Xinje XCPPro project, PLC1: XC3-24 (software 3.3L)

PROGRAM Ladder

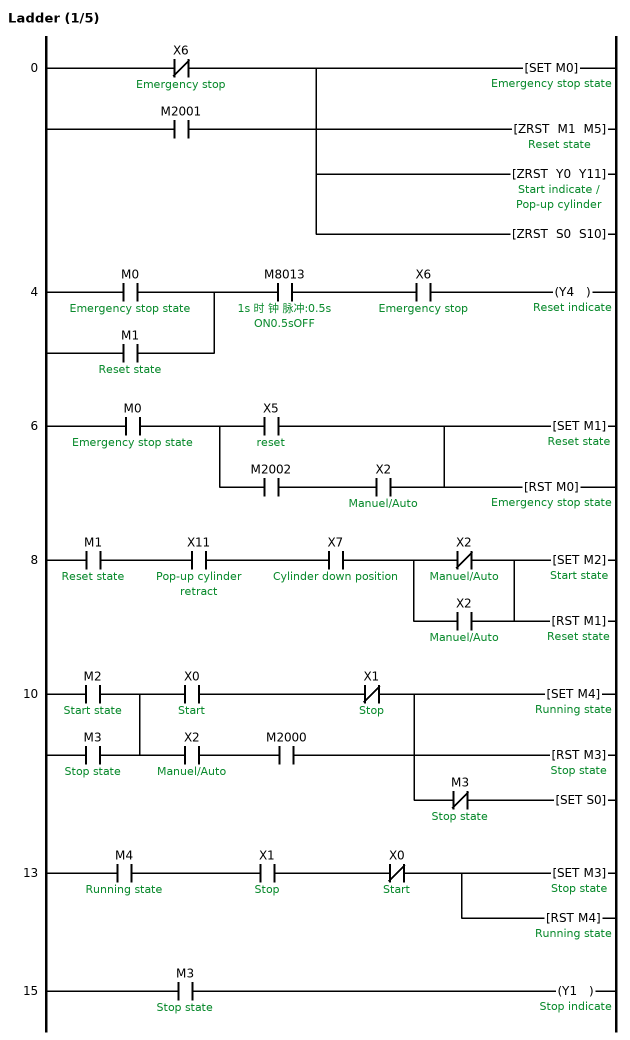
LDI    X6	; Emergency stop
OR     M2001
SET    M0	; Emergency stop state
ZRST   M1 M5	; Reset state
ZRST   Y0 Y11	; Start indicate / Pop-up cylinder
ZRST   S0 S10
LD     M0	; Emergency stop state
OR     M1	; Reset state
AND    M8013	; 1s 时 钟 脉冲:0.5s ON0.5sOFF
AND    X6	; Emergency stop
OUT    Y4	; Reset indicate 
LD     M0	; Emergency stop state
LD     X5	; reset
LD     M2002
AND    X2	; Manuel/Auto
ORB
ANB
SET    M1	; Reset state
RST    M0	; Emergency stop state
LD     M1	; Reset state
AND    X11	; Pop-up cylinder retract 
AND    X7	; Cylinder down position 
LDI    X2	; Manuel/Auto
OR     X2	; Manuel/Auto
ANB
SET    M2	; Start state
RST    M1	; Reset state
LD     M2	; Start state
OR     M3	; Stop state
LD     X0	; Start
ANI    X1	; Stop
LD     X2	; Manuel/Auto
AND    M2000
ORB
ANB
SET    M4	; Running state
RST    M3	; Stop state
ANI    M3	; Stop state
SET    S0
LD     M4	; Running state
AND    X1	; Stop
ANI    X0	; Start
SET    M3	; Stop state
RST    M4	; Running state
LD     M3	; Stop state
OUT    Y1	; Stop indicate

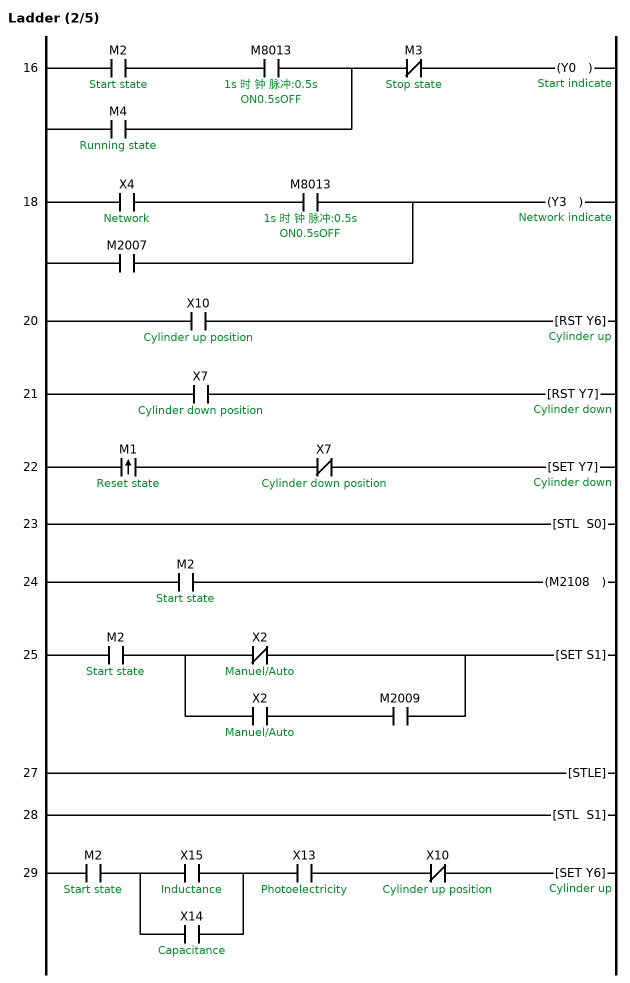
LD     M2	; Start state
AND    M8013	; 1s 时 钟 脉冲:0.5s ON0.5sOFF
OR     M4	; Running state
ANI    M3	; Stop state
OUT    Y0	; Start indicate
LD     X4	; Network
AND    M8013	; 1s 时 钟 脉冲:0.5s ON0.5sOFF
OR     M2007
OUT    Y3	; Network indicate
LD     X10	; Cylinder up position
RST    Y6	; Cylinder up 
LD     X7	; Cylinder down position 
RST    Y7	; Cylinder down
LDP    M1	; Reset state
ANI    X7	; Cylinder down position 
SET    Y7	; Cylinder down
STL    S0
LD     M2	; Start state
OUT    M2108
LD     M2	; Start state
LDI    X2	; Manuel/Auto
LD     X2	; Manuel/Auto
AND    M2009
ORB
ANB
SET    S1
STLE
STL    S1
LD     M2	; Start state
LD     X15	; Inductance
OR     X14	; Capacitance
ANB
AND    X13	; Photoelectricity
ANI    X10	; Cylinder up position
SET    Y6	; Cylinder up 

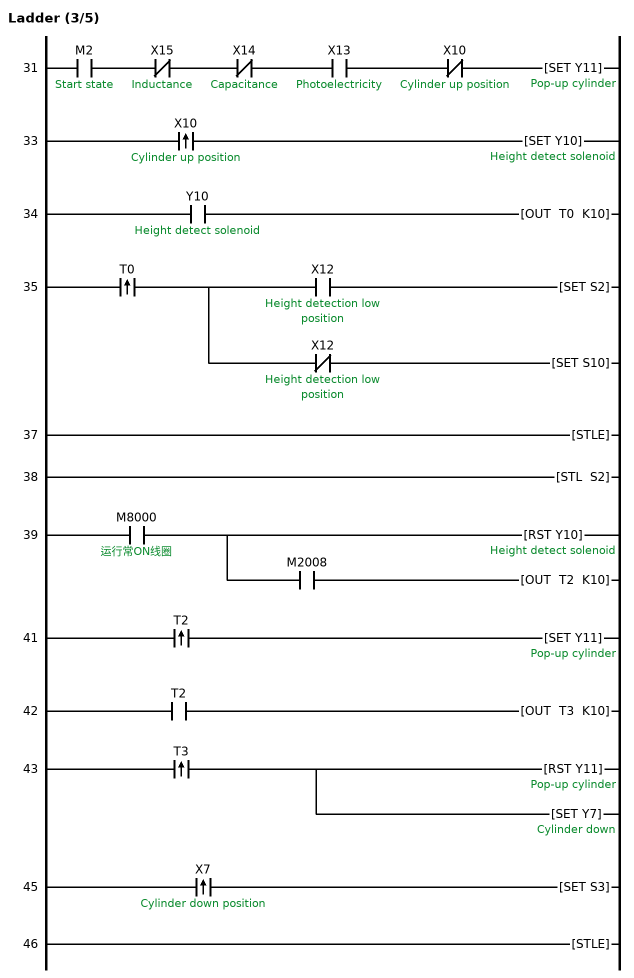
LD     M2	; Start state
ANI    X15	; Inductance
ANI    X14	; Capacitance
AND    X13	; Photoelectricity
ANI    X10	; Cylinder up position
SET    Y11	; Pop-up cylinder
LDP    X10	; Cylinder up position
SET    Y10	; Height detect solenoid
LD     Y10	; Height detect solenoid
OUT    T0 K10
LDP    T0
MPS
AND    X12	; Height detection low position
SET    S2
MPP
ANI    X12	; Height detection low position
SET    S10
STLE
STL    S2
LD     M8000	; 运行常ON线圈
RST    Y10	; Height detect solenoid
AND    M2008
OUT    T2 K10
LDP    T2
SET    Y11	; Pop-up cylinder
LD     T2
OUT    T3 K10
LDP    T3
RST    Y11	; Pop-up cylinder
SET    Y7	; Cylinder down
LDP    X7	; Cylinder down position 
SET    S3
STLE

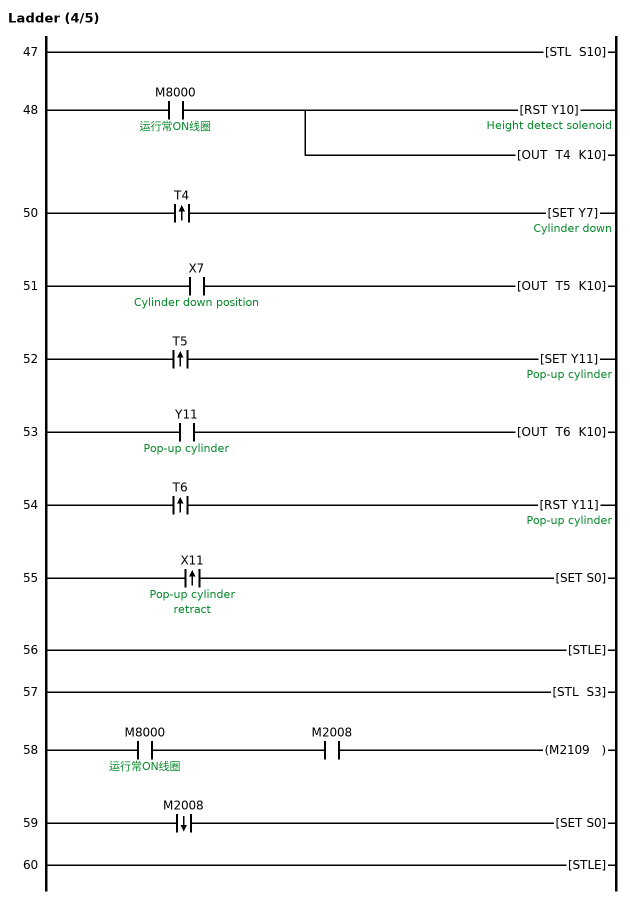
STL    S10
LD     M8000	; 运行常ON线圈
RST    Y10	; Height detect solenoid
OUT    T4 K10
LDP    T4
SET    Y7	; Cylinder down
LD     X7	; Cylinder down position 
OUT    T5 K10
LDP    T5
SET    Y11	; Pop-up cylinder
LD     Y11	; Pop-up cylinder
OUT    T6 K10
LDP    T6
RST    Y11	; Pop-up cylinder
LDP    X11	; Pop-up cylinder retract 
SET    S0
STLE
STL    S3
LD     M8000	; 运行常ON线圈
AND    M2008
OUT    M2109
LDF    M2008
SET    S0
STLE

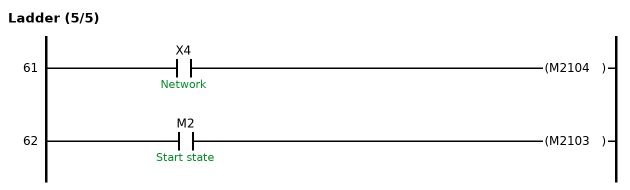
LD     X4	; Network
OUT    M2104
LD     M2	; Start state
OUT    M2103

COMMENTS (devices not used above)
X3	Height detection high position 
Y5	Alarm indicate